// TIA Portal V17 export
// export: Created 2025-05-22T05:59:44.7244498Z, ExportSetting WithDefaults, DisplayName Totally Integrated Automation Portal, DisplayVersion V17 Update 8, DisplayName TIA Portal Openness, DisplayVersion V17 Update 8, DisplayName TIA Portal Version Control Interface, DisplayVersion V17, DisplayName SINAMICS Startdrive Advanced, DisplayVersion V17 SP2, DisplayName SINAMICS Startdrive G110M, G120, G120C, G120D, G120P, G115D, DisplayVersion V17 SP2, DisplayName SINAMICS Startdrive G130, G150, S120, S150, SINAMICS MV, S210, DisplayVersion V17 SP2, DisplayName STEP 7 Professional, DisplayVersion V17 Update 8, DisplayName SINUMERIK ONE STEP 7 Toolbox, DisplayVersion V17 Update 12, DisplayName SINUMERIK ONE PLC Basic Program Plus, DisplayVersion V17 Update 12, DisplayName SINUMERIK 840D sl STEP 7 Toolbox, DisplayVersion V17 Update 12, DisplayName STEP 7 Safety, DisplayVersion V17 Update 6, DisplayName WinCC Advanced, DisplayVersion V17 Update 8
FUNCTION "FC7320_ROBOT_CELL_INTERLOCK" : Void   // FC7320, LAD
{ S7_Optimized_Access := 'FALSE' }
AUTHOR : ETXETAR
VERSION : 1.0
// stored: AutoNumber false, IsIECCheckEnabled false, SetENOAutomatically false, UDAEnableTagReadback false
   VAR_TEMP
      INPUTS_UNIT_01 : HW_IO;
      INPUTS_UNIT_02 : HW_IO;
      OUTPUTS_UNIT_01 : HW_IO;
      OUTPUTS_UNIT_02 : HW_IO;
      RETVAL_FILL : Int;
   END_VAR
   VAR_TEMP   // added for the SCL form of the ladder/FBD networks
      _w1 : Bool;
   END_VAR
BEGIN

REGION Network 1: INPUTS
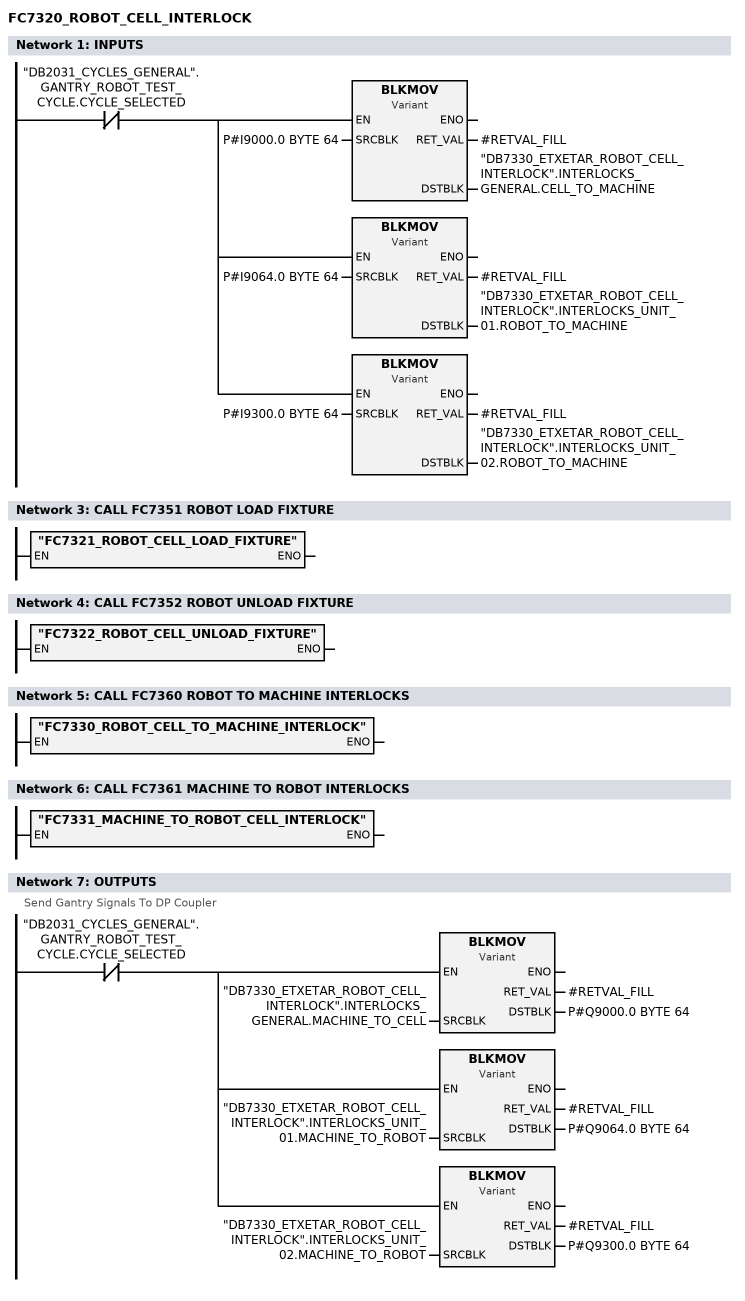
   RUNG wire#powerrail
      I_Contact( "DB2031_CYCLES_GENERAL".GANTRY_ROBOT_TEST_CYCLE.CYCLE_SELECTED )
      wire#w1
      { S7_Templates := "blk_type := Variant" } BLKMOV(SRCBLK := P#I9000.0 BYTE 64, RET_VAL => #RETVAL_FILL, DSTBLK => "DB7330_ETXETAR_ROBOT_CELL_INTERLOCK".INTERLOCKS_GENERAL.CELL_TO_MACHINE)
   END_RUNG
   RUNG wire#w1
      { S7_Templates := "blk_type := Variant" } BLKMOV(SRCBLK := P#I9064.0 BYTE 64, RET_VAL => #RETVAL_FILL, DSTBLK => "DB7330_ETXETAR_ROBOT_CELL_INTERLOCK".INTERLOCKS_UNIT_01.ROBOT_TO_MACHINE)
   END_RUNG
   RUNG wire#w1
      { S7_Templates := "blk_type := Variant" } BLKMOV(SRCBLK := P#I9300.0 BYTE 64, RET_VAL => #RETVAL_FILL, DSTBLK => "DB7330_ETXETAR_ROBOT_CELL_INTERLOCK".INTERLOCKS_UNIT_02.ROBOT_TO_MACHINE)
   END_RUNG
   // the same network as SCL:
   #_w1 := NOT "DB2031_CYCLES_GENERAL".GANTRY_ROBOT_TEST_CYCLE.CYCLE_SELECTED;
   IF #_w1 THEN
       #RETVAL_FILL := BLKMOV(SRCBLK := P#I9000.0 BYTE 64,
                              DSTBLK => "DB7330_ETXETAR_ROBOT_CELL_INTERLOCK".INTERLOCKS_GENERAL.CELL_TO_MACHINE);
       #RETVAL_FILL := BLKMOV(SRCBLK := P#I9064.0 BYTE 64,
                              DSTBLK => "DB7330_ETXETAR_ROBOT_CELL_INTERLOCK".INTERLOCKS_UNIT_01.ROBOT_TO_MACHINE);
       #RETVAL_FILL := BLKMOV(SRCBLK := P#I9300.0 BYTE 64,
                              DSTBLK => "DB7330_ETXETAR_ROBOT_CELL_INTERLOCK".INTERLOCKS_UNIT_02.ROBOT_TO_MACHINE);
   END_IF;
END_REGION

REGION Network 3: CALL FC7351 ROBOT LOAD FIXTURE
   RUNG wire#powerrail
      "FC7321_ROBOT_CELL_LOAD_FIXTURE"()
   END_RUNG
   // the same network as SCL:
   "FC7321_ROBOT_CELL_LOAD_FIXTURE"();
END_REGION

REGION Network 4: CALL FC7352 ROBOT UNLOAD FIXTURE
   RUNG wire#powerrail
      "FC7322_ROBOT_CELL_UNLOAD_FIXTURE"()
   END_RUNG
   // the same network as SCL:
   "FC7322_ROBOT_CELL_UNLOAD_FIXTURE"();
END_REGION

REGION Network 5: CALL FC7360 ROBOT TO MACHINE INTERLOCKS
   RUNG wire#powerrail
      "FC7330_ROBOT_CELL_TO_MACHINE_INTERLOCK"()
   END_RUNG
   // the same network as SCL:
   "FC7330_ROBOT_CELL_TO_MACHINE_INTERLOCK"();
END_REGION

REGION Network 6: CALL FC7361 MACHINE TO ROBOT INTERLOCKS
   RUNG wire#powerrail
      "FC7331_MACHINE_TO_ROBOT_CELL_INTERLOCK"()
   END_RUNG
   // the same network as SCL:
   "FC7331_MACHINE_TO_ROBOT_CELL_INTERLOCK"();
END_REGION

REGION Network 7: OUTPUTS
   // Send Gantry Signals To DP Coupler
   RUNG wire#powerrail
      I_Contact( "DB2031_CYCLES_GENERAL".GANTRY_ROBOT_TEST_CYCLE.CYCLE_SELECTED )
      wire#w1
      { S7_Templates := "blk_type := Variant" } BLKMOV(SRCBLK := "DB7330_ETXETAR_ROBOT_CELL_INTERLOCK".INTERLOCKS_GENERAL.MACHINE_TO_CELL, RET_VAL => #RETVAL_FILL, DSTBLK => P#Q9000.0 BYTE 64)
   END_RUNG
   RUNG wire#w1
      { S7_Templates := "blk_type := Variant" } BLKMOV(SRCBLK := "DB7330_ETXETAR_ROBOT_CELL_INTERLOCK".INTERLOCKS_UNIT_01.MACHINE_TO_ROBOT, RET_VAL => #RETVAL_FILL, DSTBLK => P#Q9064.0 BYTE 64)
   END_RUNG
   RUNG wire#w1
      { S7_Templates := "blk_type := Variant" } BLKMOV(SRCBLK := "DB7330_ETXETAR_ROBOT_CELL_INTERLOCK".INTERLOCKS_UNIT_02.MACHINE_TO_ROBOT, RET_VAL => #RETVAL_FILL, DSTBLK => P#Q9300.0 BYTE 64)
   END_RUNG
   // the same network as SCL:
   #_w1 := NOT "DB2031_CYCLES_GENERAL".GANTRY_ROBOT_TEST_CYCLE.CYCLE_SELECTED;
   IF #_w1 THEN
       #RETVAL_FILL := BLKMOV(SRCBLK := "DB7330_ETXETAR_ROBOT_CELL_INTERLOCK".INTERLOCKS_GENERAL.MACHINE_TO_CELL,
                              DSTBLK => P#Q9000.0 BYTE 64);
       #RETVAL_FILL := BLKMOV(SRCBLK := "DB7330_ETXETAR_ROBOT_CELL_INTERLOCK".INTERLOCKS_UNIT_01.MACHINE_TO_ROBOT,
                              DSTBLK => P#Q9064.0 BYTE 64);
       #RETVAL_FILL := BLKMOV(SRCBLK := "DB7330_ETXETAR_ROBOT_CELL_INTERLOCK".INTERLOCKS_UNIT_02.MACHINE_TO_ROBOT,
                              DSTBLK => P#Q9300.0 BYTE 64);
   END_IF;
END_REGION
END_FUNCTION
